(* Logix 5000 project; controller FactoryIO Emulate 5570 rev 33.11; software revision 33.00 *)

TASK MainTask (continuous, watchdog 500 ms) : MainProgram

MODULES
   Local : Emulate 5570 (ICP 2, rev 33.11)
END_MODULES

TYPE Box_Pick :
STRUCT
   X : REAL;
   Y : REAL;
   Z : REAL;
END_STRUCT
END_TYPE

TYPE Box_Place :
STRUCT
   X : REAL;
   Y : REAL;
   Z : REAL;
   C_Pos : BOOL;
END_STRUCT
END_TYPE

VAR_GLOBAL   (* controller tags *)
   At_PickUp : BOOL;
   At_Pickup_Timer : FBD_TIMER := (PRE := 600);
   At_PickUpAppro : BOOL;
   At_PickUpAppro_Timer : FBD_TIMER := (PRE := 600);
   At_Place_Box : BOOL;
   At_Place_Box_Appro : BOOL;
   At_Place_Box_Appro_Timer : FBD_TIMER := (PRE := 600);
   At_Place_Box_Timer : FBD_TIMER := (PRE := 600);
   Auto : ALIAS FOR BOOL_IN_8;
   BOOL_IN_0 : BOOL := 1;
   BOOL_IN_1 : BOOL := 1;
   BOOL_IN_10 : BOOL := 1;
   BOOL_IN_11 : BOOL := 1;
   BOOL_IN_12 : BOOL := 1;
   BOOL_IN_2 : BOOL;
   BOOL_IN_3 : BOOL := 1;
   BOOL_IN_4 : BOOL;
   BOOL_IN_5 : BOOL;
   BOOL_IN_6 : BOOL := 1;
   BOOL_IN_7 : BOOL := 1;
   BOOL_IN_8 : BOOL;
   BOOL_IN_9 : BOOL;
   BOOL_OUT_0 : BOOL;
   BOOL_OUT_1 : BOOL;
   BOOL_OUT_10 : BOOL;
   BOOL_OUT_2 : BOOL;
   BOOL_OUT_3 : BOOL;
   BOOL_OUT_4 : BOOL;
   BOOL_OUT_5 : BOOL;
   BOOL_OUT_6 : BOOL := 1;
   BOOL_OUT_7 : BOOL := 1;
   BOOL_OUT_8 : BOOL;
   BOOL_OUT_9 : BOOL := 1;
   Box_At_Place : ALIAS FOR BOOL_IN_0;
   Box_At_Place_Falling_Edge : BOOL;
   Box_At_Place_Storage_Bit : BOOL := 1;
   Box_Conveyor : ALIAS FOR BOOL_OUT_0;
   Box_Conveyor_Flags : BOOL[32] := ([0] := 1);
   Box_Conveyor_Step_Number : INT;
   Box_Pick : Box_Pick := (X := 8.0, Y := 5.5, Z := 5.2); {constant}
   Box_Place : Box_Place[6] := ([0].X := 3.2, [0].Y := 3.4, [0].Z := 10.0, [1].X := 3.2, [1].Y := 6.4, [1].Z := 10.0, [2].X := 2.5, [2].Y := 4.8, [2].Z := 5.5, [2].C_Pos := 1, [3].X := 4.2, [3].Y := 4.8, [3].Z := 5.5, [3].C_Pos := 1, [4].X := 3.2, [4].Y := 3.4, [4].Z := 1.0, [5].X := 3.2, [5].Y := 6.4, [5].Z := 1.0); {constant}
   C : ALIAS FOR BOOL_OUT_3;
   C_Limit : ALIAS FOR BOOL_IN_3;
   Call_Next_Box : BOOL;
   Cartesian_Step_Number : INT;
   Counter : ALIAS FOR INT_OUT_0;
   Delay_Time : DINT := 600; {constant}
   Detected : ALIAS FOR BOOL_IN_2;
   Emergency_OK : BOOL;
   Emergency_Stop : ALIAS FOR BOOL_IN_7;
   Exit_Conveyor : ALIAS FOR BOOL_OUT_2;
   Exit_Conveyor_End : ALIAS FOR BOOL_IN_11;
   Exit_Conveyor_End_Rising_Edge : BOOL;
   Exit_Conveyor_End_Storage_Bit : BOOL := 1;
   Exit_Conveyor_Entry : ALIAS FOR BOOL_IN_10;
   Exit_Conveyor_Flags : BOOL[32];
   Exit_Green_Lamp : ALIAS FOR BOOL_OUT_5;
   Exit_Red_Lamp : ALIAS FOR BOOL_OUT_7;
   Exit_Yellow_Lamp : ALIAS FOR BOOL_OUT_6;
   Factory_IO_CameraPosition : ALIAS FOR INT_OUT_1;
   Factory_IO_Running : ALIAS FOR BOOL_IN_9;
   FALSE : BOOL;
   Flasher : BOOL := 1;
   flip : TIMER := (PRE := 500, ACC := 500, EN := 1, DN := 1);
   FLOAT_IN_0 : REAL;
   FLOAT_IN_1 : REAL;
   FLOAT_IN_2 : REAL;
   FLOAT_OUT_0 : REAL;
   FLOAT_OUT_1 : REAL;
   FLOAT_OUT_2 : REAL;
   flop : TIMER := (PRE := 500, ACC := 347, EN := 1, TT := 1);
   Goto_PickUp : BOOL;
   Goto_PickUpAppro : BOOL;
   Goto_PlaceBox : BOOL;
   Goto_PlaceBox_Appro : BOOL;
   Grab : ALIAS FOR BOOL_OUT_4;
   INT_OUT_0 : DINT;
   INT_OUT_1 : DINT;
   Manual : ALIAS FOR BOOL_IN_12;
   Part_At_Place : ALIAS FOR BOOL_IN_1;
   Part_Conveyor : ALIAS FOR BOOL_OUT_1;
   Reset : ALIAS FOR BOOL_IN_5;
   Reset_Light : ALIAS FOR BOOL_OUT_9;
   Reset_System : BOOL;
   SP_X : ALIAS FOR FLOAT_OUT_0;
   SP_Y : ALIAS FOR FLOAT_OUT_1;
   SP_Z : ALIAS FOR FLOAT_OUT_2;
   Start : ALIAS FOR BOOL_IN_4;
   Start_Light : ALIAS FOR BOOL_OUT_8;
   Stop : ALIAS FOR BOOL_IN_6;
   Stop_Light : ALIAS FOR BOOL_OUT_10;
   System_Started : BOOL;
   Timer_CamPos : TIMER := (PRE := 5000);
   timer_grab : TIMER := (PRE := 200);
   TRUE : BOOL := 1;
   X : ALIAS FOR FLOAT_IN_0;
   X_Rounded : REAL;
   Y : ALIAS FOR FLOAT_IN_1;
   Y_Rounded : REAL;
   Z : ALIAS FOR FLOAT_OUT_2;
   Z_Rounded : REAL;
END_VAR

PROGRAM MainProgram   (* main routine MainRoutine *)
VAR
   Box_Place_Index : INT;
END_VAR

ROUTINE Camera_Positions   (* ladder *)
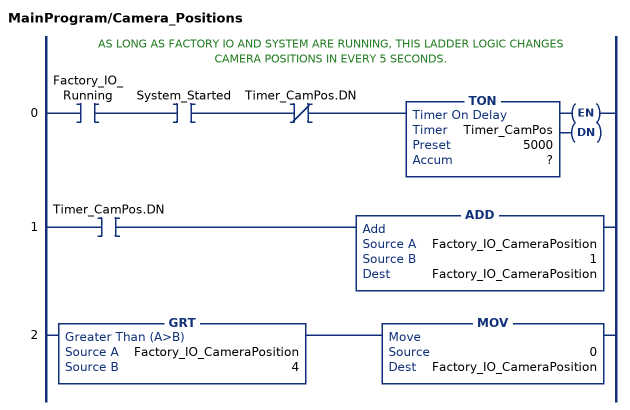
   // AS LONG AS FACTORY IO AND SYSTEM ARE RUNNING, THIS LADDER LOGIC CHANGES CAMERA POSITIONS IN EVERY 5 SECONDS.
   0: XIC(Factory_IO_Running)XIC(System_Started)XIO(Timer_CamPos.DN)TON(Timer_CamPos,?,?);
   1: XIC(Timer_CamPos.DN)ADD(Factory_IO_CameraPosition,1,Factory_IO_CameraPosition);
   2: GRT(Factory_IO_CameraPosition,4)MOV(0,Factory_IO_CameraPosition);
END_ROUTINE

ROUTINE Cartesian   (* ladder *)
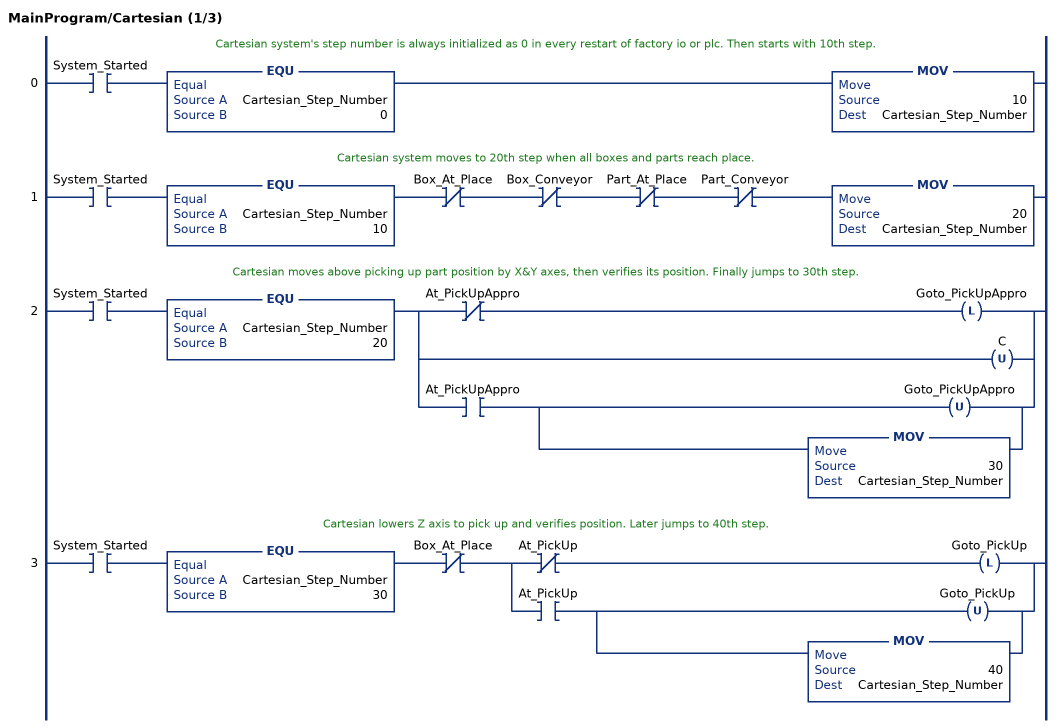
   // Cartesian system's step number is always initialized as 0 in every restart of factory io or plc. Then starts with 10th step.
   0: XIC(System_Started)EQU(Cartesian_Step_Number,0)MOV(10,Cartesian_Step_Number);
   // Cartesian system moves to 20th step when all boxes and parts reach place.
   1: XIC(System_Started)EQU(Cartesian_Step_Number,10)XIO(Box_At_Place)XIO(Box_Conveyor)XIO(Part_At_Place)XIO(Part_Conveyor)MOV(20,Cartesian_Step_Number);
   // Cartesian moves above picking up part position by X&Y axes, then verifies its position. Finally jumps to 30th step.
   2: XIC(System_Started)EQU(Cartesian_Step_Number,20)[[XIO(At_PickUpAppro) OTL(Goto_PickUpAppro) ,OTU(C) ] ,XIC(At_PickUpAppro) [OTU(Goto_PickUpAppro) ,MOV(30,Cartesian_Step_Number) ] ];
   // Cartesian lowers Z axis to pick up and verifies position. Later jumps to 40th step.
   3: XIC(System_Started)EQU(Cartesian_Step_Number,30)XIO(Box_At_Place)[XIO(At_PickUp) OTL(Goto_PickUp) ,XIC(At_PickUp) [OTU(Goto_PickUp) ,MOV(40,Cartesian_Step_Number) ] ];
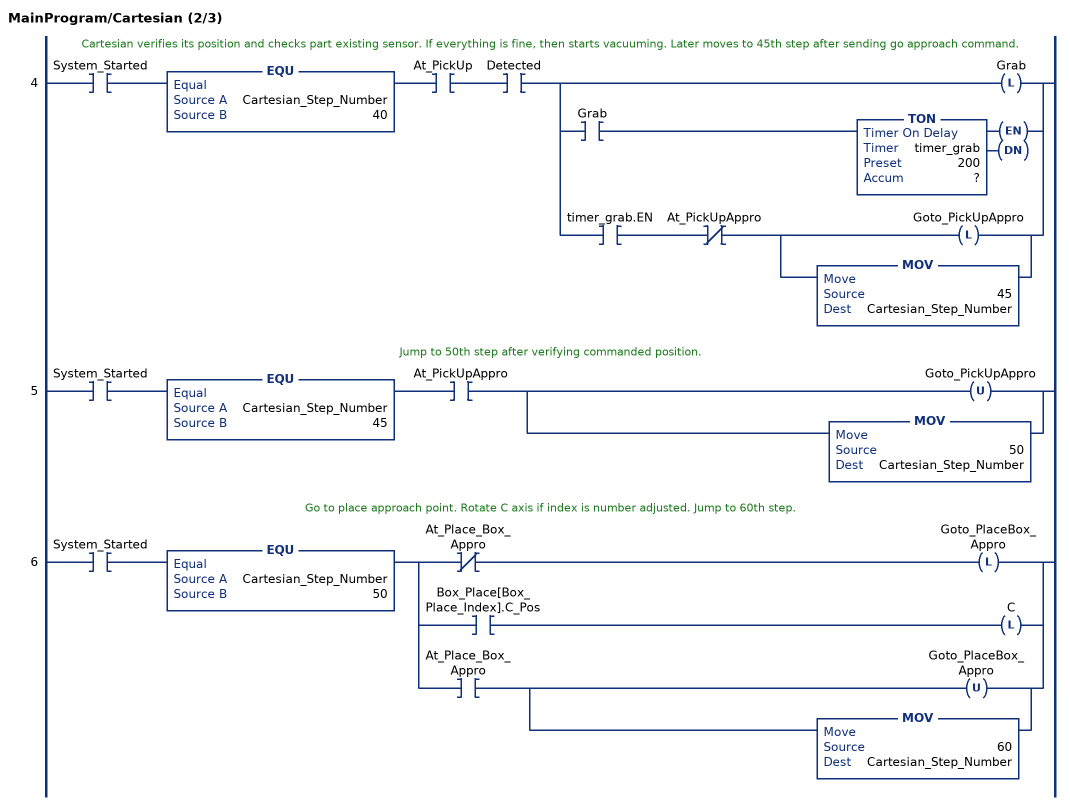
   // Cartesian verifies its position and checks part existing sensor. If everything is fine, then starts vacuuming. Later moves to 45th step after sending go approach command.
   4: XIC(System_Started)EQU(Cartesian_Step_Number,40)XIC(At_PickUp)XIC(Detected)[OTL(Grab) ,[XIC(Grab) TON(timer_grab,?,?) ,XIC(timer_grab.EN) XIO(At_PickUpAppro) [OTL(Goto_PickUpAppro) ,MOV(45,Cartesian_Step_Number) ] ] ];
   // Jump to 50th step after verifying commanded position.
   5: XIC(System_Started)EQU(Cartesian_Step_Number,45)XIC(At_PickUpAppro)[OTU(Goto_PickUpAppro) ,MOV(50,Cartesian_Step_Number) ];
   // Go to place approach point. Rotate C axis if index is number adjusted. Jump to 60th step.
   6: XIC(System_Started)EQU(Cartesian_Step_Number,50)[[XIO(At_Place_Box_Appro) OTL(Goto_PlaceBox_Appro) ,XIC(Box_Place[Box_Place_Index].C_Pos) OTL(C) ] ,XIC(At_Place_Box_Appro) [OTU(Goto_PlaceBox_Appro) ,MOV(60,Cartesian_Step_Number) ] ];
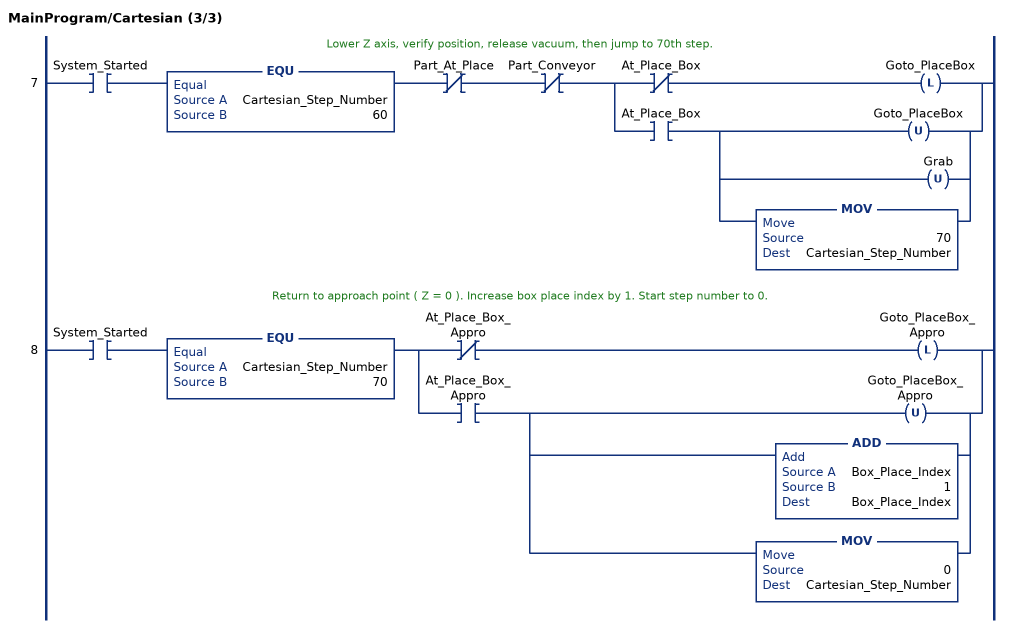
   // Lower Z axis, verify position, release vacuum, then jump to 70th step.
   7: XIC(System_Started)EQU(Cartesian_Step_Number,60)XIO(Part_At_Place)XIO(Part_Conveyor)[XIO(At_Place_Box) OTL(Goto_PlaceBox) ,XIC(At_Place_Box) [[OTU(Goto_PlaceBox) ,OTU(Grab) ] ,MOV(70,Cartesian_Step_Number) ] ];
   // Return to approach point ( Z = 0 ). Increase box place index by 1. Start step number to 0.
   8: XIC(System_Started)EQU(Cartesian_Step_Number,70)[XIO(At_Place_Box_Appro) OTL(Goto_PlaceBox_Appro) ,XIC(At_Place_Box_Appro) [OTU(Goto_PlaceBox_Appro) ,[ADD(Box_Place_Index,1,Box_Place_Index) ,MOV(0,Cartesian_Step_Number) ] ] ];
END_ROUTINE

ROUTINE Cartesian_Positions   (* structured text *)
   //Round X,Y,Z values. Values from factory io are not received rounded. A little math trick is required to round them.
   X_Rounded := (TRUNC((X*100)+0.5))/100;
   Y_Rounded := (TRUNC((Y*100)+0.5))/100;
   Z_Rounded := (TRUNC((Z*100)+0.5))/100;
   
   //Box pick positions
   
   if Goto_PickUp then
   	SP_X := Box_Pick.X;
   	SP_Y := Box_Pick.Y;
   	SP_Z := Box_Pick.Z;
   end_if;
   
   if Goto_PickUpAppro then
   	SP_X := Box_Pick.X;
   	SP_Y := Box_Pick.Y;
   	SP_Z := 0.0;
   end_if;
   
   //Verifying picking up positions. Timers are used.
   
   TONR(At_Pickup_Timer);
   At_Pickup_Timer.PRE := Delay_Time;
   At_Pickup_Timer.TimerEnable := (Box_Pick.X = X_Rounded) AND (Box_Pick.Y = Y_Rounded) AND (Box_Pick.Z = Z_Rounded);
   if At_Pickup_Timer.DN then
   	At_PickUp := TRUE;
   else
   	At_PickUp := FALSE;
   end_if;
   
   TONR(At_PickUpAppro_Timer);
   At_PickUpAppro_Timer.PRE := Delay_Time;
   At_PickUpAppro_Timer.TimerEnable := (Box_Pick.X = X_Rounded) AND (Box_Pick.Y = Y_Rounded) AND (0.0 = Z_Rounded);
   if At_PickUpAppro_Timer.DN then
   	At_PickUpAppro := TRUE;
   else
   	At_PickUpAppro := FALSE;
   end_if;
   
   // If Box Place Index is larger than 5, reset to 0. Call next box plate.
   if Box_Place_Index>=6 then
   	Box_Place_Index:=0;
   	Call_Next_Box := TRUE;
   end_if;
   
   //Box place positions.
   
   if Goto_PlaceBox then
   	SP_X := Box_Place[Box_Place_Index].X;
   	SP_Y := Box_Place[Box_Place_Index].Y;
   	SP_Z := Box_Place[Box_Place_Index].Z;
   end_if;
   
   if Goto_PlaceBox_Appro then
   	SP_X := Box_Place[Box_Place_Index].X;
   	SP_Y := Box_Place[Box_Place_Index].Y;
   	SP_Z := 0.0;
   end_if;
   
   //Verifying placing box positions. Timers are used.
   
   TONR(At_Place_Box_Timer);
   At_Place_Box_Timer.PRE := Delay_Time;
   At_Place_Box_Timer.TimerEnable := (Box_Place[Box_Place_Index].X=X_Rounded) AND (Box_Place[Box_Place_Index].Y=Y_Rounded) AND (Box_Place[Box_Place_Index].Z=Z_Rounded);
   if At_Place_Box_Timer.DN then
   	At_Place_Box := TRUE;
   else
   	At_Place_Box := FALSE;
   end_if;
   
   TONR(At_Place_Box_Appro_Timer);
   At_Place_Box_Appro_Timer.PRE := Delay_Time;
   At_Place_Box_Appro_Timer.TimerEnable := (Box_Place[Box_Place_Index].X=X_Rounded) AND (Box_Place[Box_Place_Index].Y=Y_Rounded) AND (0.0=Z_Rounded);
   if At_Place_Box_Appro_Timer.DN then
   	At_Place_Box_Appro := TRUE;
   else
   	At_Place_Box_Appro := FALSE;
   end_if;
   
END_ROUTINE

ROUTINE Conveyor_Box   (* ladder *)
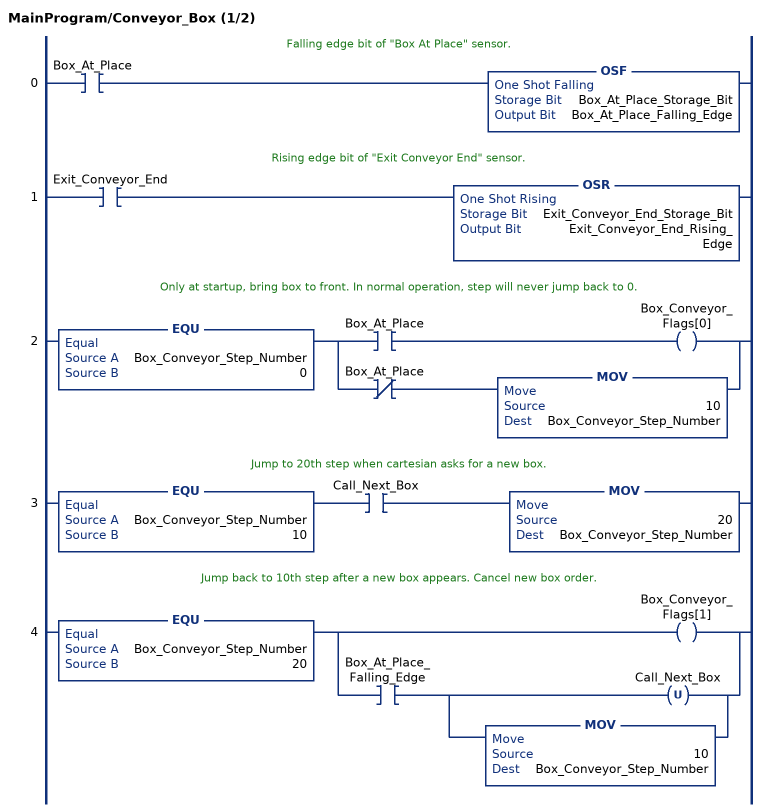
   // Falling edge bit of "Box At Place" sensor.
   0: XIC(Box_At_Place)OSF(Box_At_Place_Storage_Bit,Box_At_Place_Falling_Edge);
   // Rising edge bit of "Exit Conveyor End" sensor.
   1: XIC(Exit_Conveyor_End)OSR(Exit_Conveyor_End_Storage_Bit,Exit_Conveyor_End_Rising_Edge);
   // Only at startup, bring box to front. In normal operation, step will never jump back to 0.
   2: EQU(Box_Conveyor_Step_Number,0)[XIC(Box_At_Place) OTE(Box_Conveyor_Flags[0]) ,XIO(Box_At_Place) MOV(10,Box_Conveyor_Step_Number) ];
   // Jump to 20th step when cartesian asks for a new box.
   3: EQU(Box_Conveyor_Step_Number,10)XIC(Call_Next_Box)MOV(20,Box_Conveyor_Step_Number);
   // Jump back to 10th step after a new box appears. Cancel new box order.
   4: EQU(Box_Conveyor_Step_Number,20)[OTE(Box_Conveyor_Flags[1]) ,XIC(Box_At_Place_Falling_Edge) [OTU(Call_Next_Box) ,MOV(10,Box_Conveyor_Step_Number) ] ];
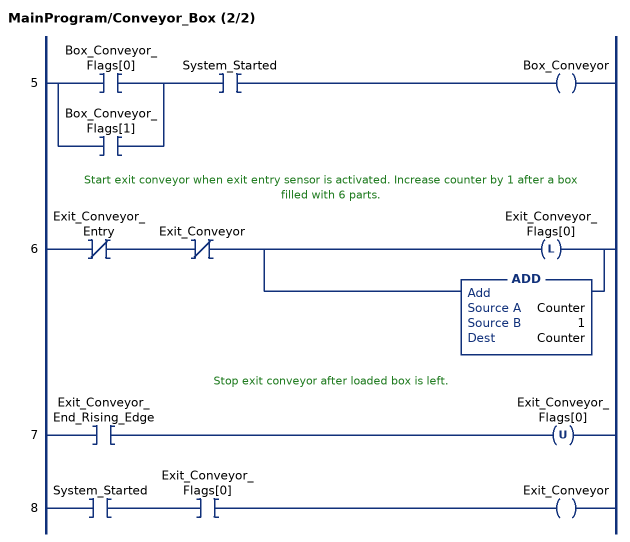
   5: [XIC(Box_Conveyor_Flags[0]) ,XIC(Box_Conveyor_Flags[1]) ]XIC(System_Started)OTE(Box_Conveyor);
   // Start exit conveyor when exit entry sensor is activated. Increase counter by 1 after a box filled with 6 parts.
   6: XIO(Exit_Conveyor_Entry)XIO(Exit_Conveyor)[OTL(Exit_Conveyor_Flags[0]) ,ADD(Counter,1,Counter) ];
   // Stop exit conveyor after loaded box is left.
   7: XIC(Exit_Conveyor_End_Rising_Edge)OTU(Exit_Conveyor_Flags[0]);
   8: XIC(System_Started)XIC(Exit_Conveyor_Flags[0])OTE(Exit_Conveyor);
END_ROUTINE

ROUTINE Conveyor_Part   (* ladder *)
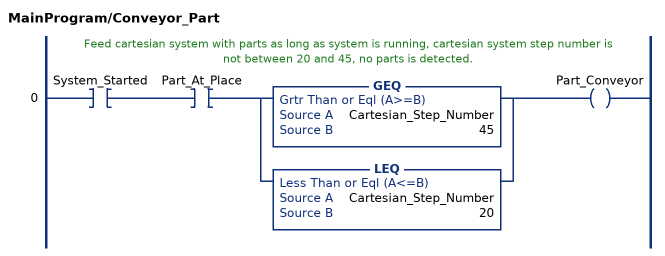
   // Feed cartesian system with parts as long as system is running, cartesian system step number is not between 20 and 45, no parts is detected.
   0: XIC(System_Started)XIC(Part_At_Place)[GEQ(Cartesian_Step_Number,45) ,LEQ(Cartesian_Step_Number,20) ]OTE(Part_Conveyor);
END_ROUTINE

ROUTINE Electric_Board   (* ladder *)
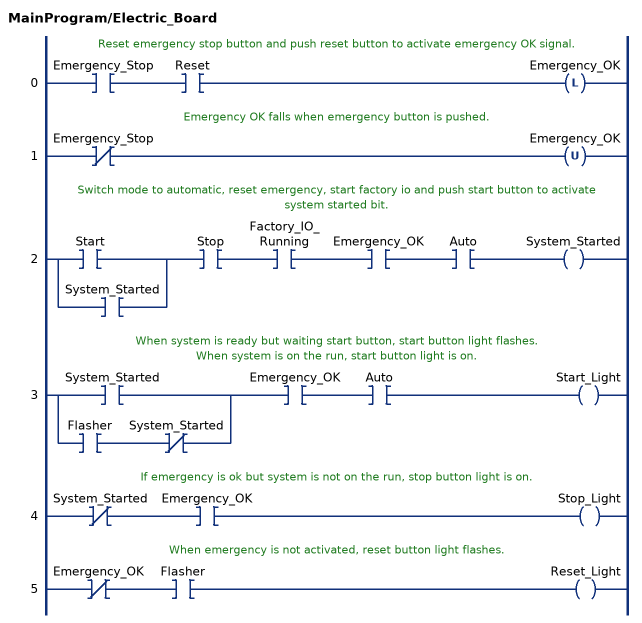
   // Reset emergency stop button and push reset button to activate emergency OK signal.
   0: XIC(Emergency_Stop)XIC(Reset)OTL(Emergency_OK);
   // Emergency OK falls when emergency button is pushed.
   1: XIO(Emergency_Stop)OTU(Emergency_OK);
   // Switch mode to automatic, reset emergency, start factory io and push start button to activate system started bit.
   2: [XIC(Start) ,XIC(System_Started) ]XIC(Stop)XIC(Factory_IO_Running)XIC(Emergency_OK)XIC(Auto)OTE(System_Started);
   // When system is ready but waiting start button, start button light flashes.
   // When system is on the run, start button light is on.
   3: [XIC(System_Started) ,XIC(Flasher) XIO(System_Started) ]XIC(Emergency_OK)XIC(Auto)OTE(Start_Light);
   // If emergency is ok but system is not on the run, stop button light is on.
   4: XIO(System_Started)XIC(Emergency_OK)OTE(Stop_Light);
   // When emergency is not activated, reset button light flashes.
   5: XIO(Emergency_OK)XIC(Flasher)OTE(Reset_Light);
END_ROUTINE

ROUTINE General   (* structured text *)
   // If factory io is not working, initialize everything.
   if not Factory_IO_Running then
   	Cartesian_Step_Number := 0;
   	Box_Conveyor_Step_Number := 0;
   	SP_X := 0.0;
   	SP_Y := 0.0;
   	SP_Z := 0.0;
   	X := 0.0;
   	Y := 0.0;
   	Z := 0.0;
   	Box_Place_Index := 0;
   	Counter := 0;
   	Factory_IO_CameraPosition := 0;
   	Grab := FALSE;
   	C := FALSE;
   	Goto_PickUp := FALSE;
   	Goto_PickUpAppro := FALSE;
   	Goto_PlaceBox := FALSE;
   	Goto_PlaceBox_Appro := FALSE;
   	Call_Next_Box := FALSE;
   	Exit_Conveyor := FALSE;
   	Emergency_OK := FALSE;
   end_if;
   
   
END_ROUTINE

ROUTINE MainRoutine   (* ladder *)
// Main function of the plc program which calls functions and involves basic logics.
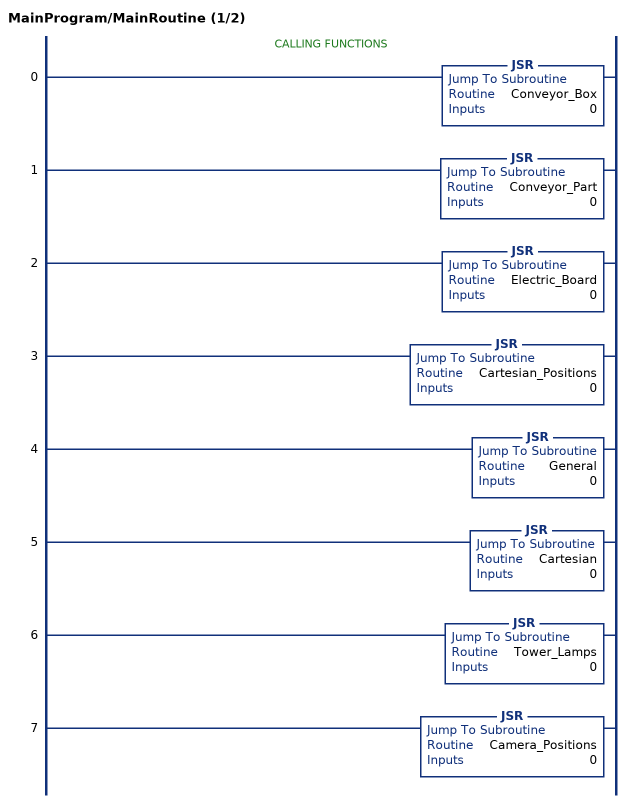
   // CALLING FUNCTIONS
   0: JSR(Conveyor_Box,0);
   1: JSR(Conveyor_Part,0);
   2: JSR(Electric_Board,0);
   3: JSR(Cartesian_Positions,0);
   4: JSR(General,0);
   5: JSR(Cartesian,0);
   6: JSR(Tower_Lamps,0);
   7: JSR(Camera_Positions,0);
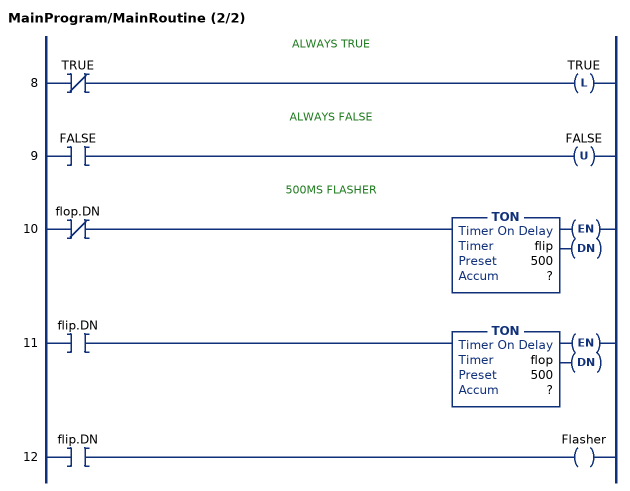
   // ALWAYS TRUE
   8: XIO(TRUE)OTL(TRUE);
   // ALWAYS FALSE
   9: XIC(FALSE)OTU(FALSE);
   // 500MS FLASHER
   10: XIO(flop.DN)TON(flip,?,?);
   11: XIC(flip.DN)TON(flop,?,?);
   12: XIC(flip.DN)OTE(Flasher);
END_ROUTINE

ROUTINE Tower_Lamps   (* ladder *)
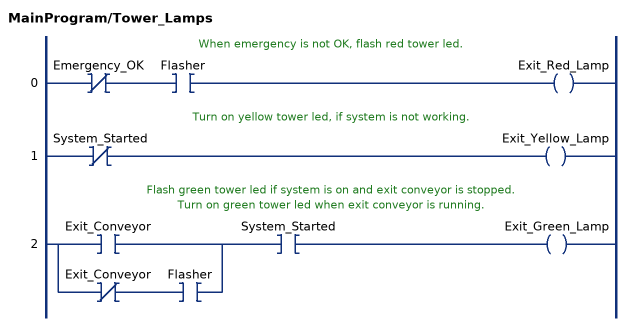
   // When emergency is not OK, flash red tower led.
   0: XIO(Emergency_OK)XIC(Flasher)OTE(Exit_Red_Lamp);
   // Turn on yellow tower led, if system is not working.
   1: XIO(System_Started)OTE(Exit_Yellow_Lamp);
   // Flash green tower led if system is on and exit conveyor is stopped.
   // Turn on green tower led when exit conveyor is running.
   2: [XIC(Exit_Conveyor) ,XIO(Exit_Conveyor) XIC(Flasher) ]XIC(System_Started)OTE(Exit_Green_Lamp);
END_ROUTINE
END_PROGRAM
